FUNCTION_BLOCK Plant
  (* Standard: 61499-2 *)
  (* Version 0.1, 2015-00-16, Th?o, PC_THEO *)
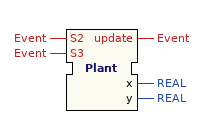
  EVENT_INPUT
    S2;
    S3;
  END_EVENT
  EVENT_OUTPUT
    update;
  END_EVENT
  VAR_OUTPUT
    x : REAL;
    y : REAL;
  END_VAR
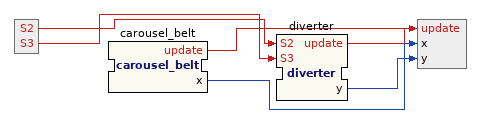
  FBS
    carousel_belt : carousel_belt;
    diverter : diverter;
  END_FBS
  EVENT_CONNECTIONS
    S2 TO diverter.S2;
    S3 TO diverter.S3;
    carousel_belt.update TO update;
    diverter.update TO update;
  END_CONNECTIONS
  DATA_CONNECTIONS
    carousel_belt.x TO x;
    diverter.y TO y;
  END_CONNECTIONS
END_FUNCTION_BLOCK
